FUNCTION_BLOCK Blinck_V2
VAR_INPUT
	Enable: BOOL;
	In_Pause: BOOL;
	Timer_Seconde_ON: REAL;
	Timer_Minute_ON: REAL;
	Timer_Heure_ON: REAL;
	Timer_Jour_ON: REAL;
	Timer_Seconde_OFF: REAL;
	Timer_Minute_OFF: REAL;
	Timer_Heure_OFF: REAL;
	Timer_Jour_OFF: REAL;
	Contact_Off: BOOL;
	Contact_On: BOOL;
END_VAR
VAR_OUTPUT
	Out: BOOL;
END_VAR
VAR
	TON_1: TON_V1;
	TON_2: TON_V1;
	Out2: BOOL;
	Out3: BOOL;
END_VAR

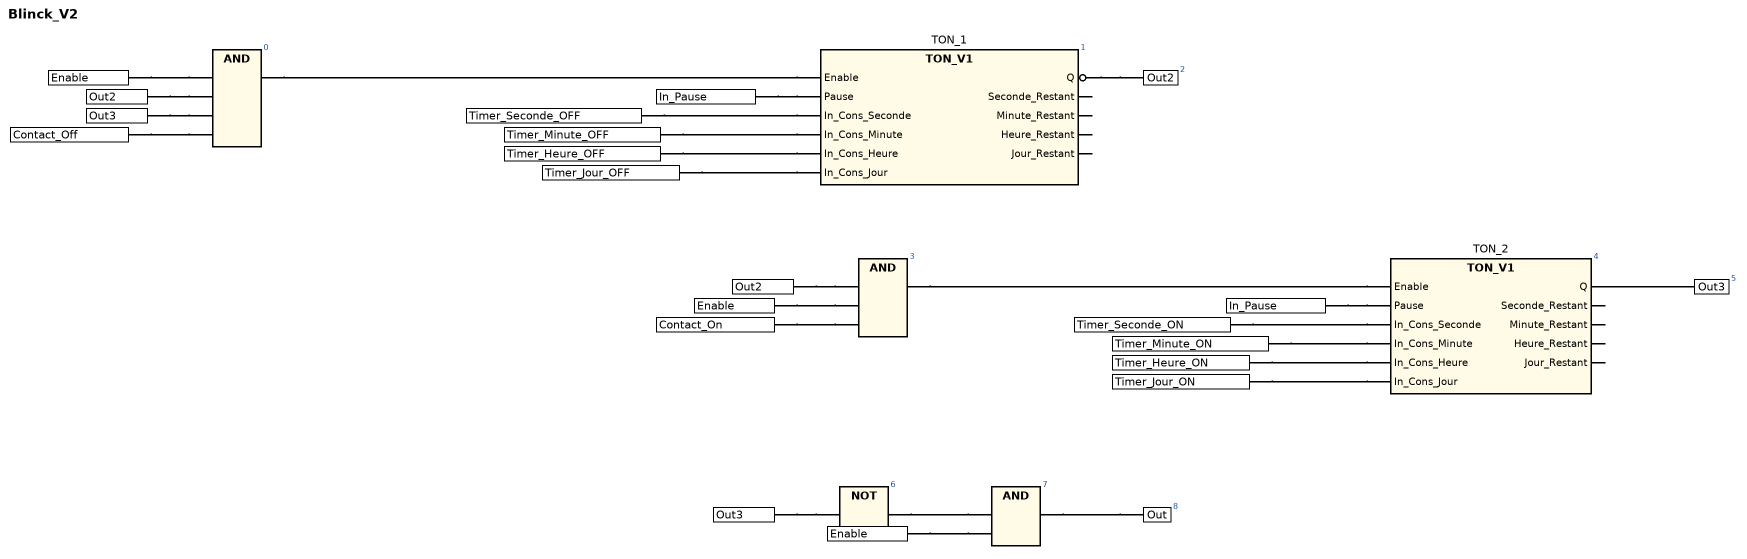
TON_1(
    Enable := Enable AND Out2 AND Out3 AND Contact_Off,
    Pause := In_Pause,
    In_Cons_Seconde := Timer_Seconde_OFF,
    In_Cons_Minute := Timer_Minute_OFF,
    In_Cons_Heure := Timer_Heure_OFF,
    In_Cons_Jour := Timer_Jour_OFF); // TON_V1
Out2 := NOT TON_1.Q;
TON_2(
    Enable := Out2 AND Enable AND Contact_On,
    Pause := In_Pause,
    In_Cons_Seconde := Timer_Seconde_ON,
    In_Cons_Minute := Timer_Minute_ON,
    In_Cons_Heure := Timer_Heure_ON,
    In_Cons_Jour := Timer_Jour_ON); // TON_V1
Out3 := TON_2.Q;
Out := NOT Out3 AND Enable;

END_FUNCTION_BLOCK

(* stored: Version 1.1.0.1, ProductVersion 3.1.4024.12
   POU Blinck_V2: Id {6ac90476-b815-47a3-9e46-c0b2ed271164}, SpecialFunc None *)
